INTERFACE I_FileWriter

METHOD WriteEvent : BOOL
VAR_INPUT
	sMessage : STRING ;
END_VAR
END_METHOD

END_INTERFACE

(* stored: Version 1.1.0.1, ProductVersion 3.1.4024.16
   Itf I_FileWriter: Id {81ac30a6-0e8a-4c0a-8dcf-fe74dce37ef3}
   Method WriteEvent: Id {88d05617-9320-4edd-83c7-6676ea1baf32} *)
